FUNCTION_BLOCK FB_DfiDbWriter_Tests EXTENDS TcUnit.FB_TestSuite
VAR
END_VAR
VAR CONSTANT
	// Espelham as constantes de FB_DfiDbWriter_Fake (VAR CONSTANT de FB nao e
	// visivel de fora da instancia). Manter os dois blocos em sincronia.
	SCRIPT_OK         : INT := 1;
	SCRIPT_EXEC_ERROR : INT := 2;
	SCRIPT_DB_LOST    : INT := 3;
END_VAR

Test_Sucesso_PopEContagem();
Test_ErroExecute_NaoPop_BackoffCresce();
Test_DbLost_DuranteExecute_VoltaIdle_SemPerder();
Test_PeriodicoTambemAtualizaBaseline();

METHOD PRIVATE Test_Sucesso_PopEContagem
VAR
	fbBuf : FB_DfiRowBuffer := (nCapacity := 8);
	sut   : FB_DfiDbWriter_Fake;   // DoExecute sempre retorna 1 (ok) apos 1 ciclo "busy"
	cfg   : ST_DfiConfig;
	r     : ST_DfiRow;
	i     : INT;
END_VAR
TEST('Sucesso_PopEContagem');
sut.SetScript(SCRIPT_OK);      // helper do fake
r.eKind := E_DfiRowKind.ESTOQUE_MUDANCA; r.stEstoque.nA := 9;
fbBuf.Push(r);
FOR i := 1 TO 20 DO sut(stConfig := cfg, fbBuffer := fbBuf); END_FOR
AssertEquals_UDINT(0, fbBuf.nCount, 'linha removida apos sucesso');
AssertEquals_ULINT(1, sut.nRowsWritten, 'nRowsWritten=1');
AssertTrue(sut.bUltimoGravadoValido, 'dedupe baseline valido');
AssertEquals_INT(9, sut.stUltimoGravado.nA, 'dedupe baseline = ultima linha de estoque');
TEST_FINISHED();
END_METHOD

METHOD PRIVATE Test_ErroExecute_NaoPop_BackoffCresce
VAR
	fbBuf : FB_DfiRowBuffer := (nCapacity := 8);
	sut   : FB_DfiDbWriter_Fake;
	cfg   : ST_DfiConfig;
	r     : ST_DfiRow;
	i     : INT;
END_VAR
TEST('ErroExecute_NaoPop');
sut.SetScript(SCRIPT_EXEC_ERROR);   // DoExecute retorna 2 (erro)
fbBuf.Push(r);
FOR i := 1 TO 30 DO sut(stConfig := cfg, fbBuffer := fbBuf); END_FOR
AssertEquals_UDINT(1, fbBuf.nCount, 'linha PRESERVADA apos erro');
AssertTrue(sut.nErrors >= 1, 'nErrors incrementa');
AssertTrue(sut.eState = E_DfiWriterState.ERROR OR sut.eState = E_DfiWriterState.IDLE, 'em ERROR/backoff ou voltando');
TEST_FINISHED();
END_METHOD

METHOD PRIVATE Test_DbLost_DuranteExecute_VoltaIdle_SemPerder
VAR
	fbBuf : FB_DfiRowBuffer := (nCapacity := 8);
	sut   : FB_DfiDbWriter_Fake;
	cfg   : ST_DfiConfig;
	r     : ST_DfiRow;
	i     : INT;
END_VAR
TEST('DbLost_SemPerder');
sut.SetScript(SCRIPT_DB_LOST);
fbBuf.Push(r);
FOR i := 1 TO 20 DO sut(stConfig := cfg, fbBuffer := fbBuf); END_FOR
AssertEquals_UDINT(1, fbBuf.nCount, 'linha preservada em DB_LOST');
TEST_FINISHED();
END_METHOD

METHOD PRIVATE Test_PeriodicoTambemAtualizaBaseline
VAR
	fbBuf : FB_DfiRowBuffer := (nCapacity := 8);
	sut   : FB_DfiDbWriter_Fake;
	cfg   : ST_DfiConfig; r : ST_DfiRow; i : INT;
END_VAR
TEST('PeriodicoAtualizaBaseline');
sut.SetScript(SCRIPT_OK);
r.eKind := E_DfiRowKind.ESTOQUE_PERIODICO; r.stEstoque.nB := 2;
fbBuf.Push(r);
FOR i := 1 TO 20 DO sut(stConfig := cfg, fbBuffer := fbBuf); END_FOR
AssertTrue(sut.bUltimoGravadoValido, 'baseline valido apos periodico');
AssertEquals_INT(2, sut.stUltimoGravado.nB, 'baseline B=2');
TEST_FINISHED();
END_METHOD

END_FUNCTION_BLOCK

(* stored: Version 1.1.0.1
   POU FB_DfiDbWriter_Tests: Id {49354fdb-87bf-4301-9321-f3075d5d6adb}, SpecialFunc None
   Method Test_Sucesso_PopEContagem: Id {12474c00-025f-45fa-bc16-a874fc2797b8}
   Method Test_ErroExecute_NaoPop_BackoffCresce: Id {6cd91532-8b0b-45b2-ba4b-8f3c2d59307b}
   Method Test_DbLost_DuranteExecute_VoltaIdle_SemPerder: Id {4b9e809f-efbd-44b7-b1cd-e0fdefe1e856}
   Method Test_PeriodicoTambemAtualizaBaseline: Id {475f70fa-1be9-4b58-8305-c4d5e443dda8} *)
